(* IEC 61131-3 sources: RL_MAR/experiments/comparison/autoplc/results/deepseek-ai-DeepSeek-V3.2_20260508_111905/med_61, 1 file *)

(* ---- med_61_3.st ---- *)
FUNCTION_BLOCK FB_Sum
VAR_INPUT
    maxValue : INT;
END_VAR
VAR_OUTPUT
    wData : WORD;
END_VAR
VAR
    II : INT;
END_VAR

    wData := 0;

    FOR II := 0 TO maxValue DO
        wData := wData + WORD_TO_INT(II);
    END_FOR;

END_FUNCTION_BLOCK
